// TwinCAT 3 PLC project CleanroomConnect
// ProgramVersion: 3.1.4024.0
// libraries:
//   KMWE Generic Library, * (KMWE)
//   Tc2_MC2, * (Beckhoff Automation GmbH)
//   Tc2_Standard, * (Beckhoff Automation GmbH)
//   Tc2_System, * (Beckhoff Automation GmbH)
//   Tc3_Module, * (Beckhoff Automation GmbH)
//   VisuDialogs, * (System)
//   VisuSymbols,3.5.10.0,System
// project tree:
//   DUTs/ I_Door.TcIO, I_AX5000.TcIO, ST_HmiBottomBar.TcDUT, ST_HmiMiddle.TcDUT, ST_HmiTopBar.TcDUT
//   / E_CtrlState.TcDUT (not stored), E_MODE.TcTLO (not stored), FB_ForceOutput.TcPOU (not stored), F_InRange.TcPOU (not stored), GlobalTextList.TcGTLO, PlcTask.TcTTO, ST_MsgBox.TcDUT (not stored)
//   GVLs/ GVL.TcGVL, GVL_Modules.TcGVL
//   POUs/02 UN/Unit %28UN%29/ ST_UN_CleanroomConnectSettings.TcDUT (not stored), UN_CleanroomConnect.TcPOU (not stored)
//   POUs/03 EM/Equipment %28EM%29/2 EM_PalletConveyor/DUT/ E_SeqCentering.TcDUT (not stored), E_ActionSelection.TcDUT (not stored), E_SeqTransport.TcDUT (not stored)
//   POUs/03 EM/Equipment %28EM%29/2 EM_PalletConveyor/ FB_ModeStateControl_PalletConveyor.TcPOU (not stored) (excluded from build), EM_PalletConveyor.TcPOU (not stored), I_EM_PalletConveyor.TcIO (not stored), ST_SettingsPalletConveyor.TcDUT (not stored)
//   POUs/03 EM/Equipment %28EM%29/4 EM_LiftingTransport/DUT/ E_SeqLiftingTransport.TcDUT (not stored), ST_PositioningProfile.TcDUT (not stored), ST_SettingsLiftingTransport.TcDUT (not stored), ST_SpeedProfile.TcDUT (not stored)
//   POUs/03 EM/Equipment %28EM%29/EM_AirTreatment/DUTs/ I_EM_AirTreatment.TcIO (not stored), ST_SettingsAirTrearment.TcDUT (not stored)
//   POUs/03 EM/Equipment %28EM%29/EM_AirTreatment/ EM_AirTreatment.TcPOU (not stored)
//   POUs/03 EM/Equipment %28EM%29/4 EM_LiftingTransport/ EM_LiftingTransport.TcPOU (not stored), I_EM_LiftingTransport.TcIO (not stored)
//   POUs/03 EM/Equipment %28EM%29/1 EM_Utilities/DUTs/ E_ForceValue.TcDUT (not stored), I_EM_Utilities.TcIO (not stored), ST_SettingsUtilities.TcDUT (not stored)
//   POUs/03 EM/Equipment %28EM%29/1 EM_Utilities/ EM_Utilities.TcPOU (not stored)
//   POUs/03 EM/Equipment %28EM%29/EM_DockingCabin/DUTs/ E_SeqDockingCabin.TcDUT (not stored), ST_SettingsDockingCabin.TcDUT (not stored)
//   POUs/03 EM/Equipment %28EM%29/EM_DockingCabin/ EM_DockingCabin.TcPOU (not stored)
//   POUs/03 EM/Equipment %28EM%29/3 EM_DockingInterface/DUTs/ E_SeqDockingInterface.TcDUT (not stored), I_EM_DockingInterface.TcIO (not stored), ST_SettingsDockingInterface.TcDUT (not stored)
//   POUs/03 EM/Equipment %28EM%29/3 EM_DockingInterface/ EM_DockingInterface.TcPOU (not stored)
//   POUs/03 EM/Equipment %28EM%29/EM_Doors/DUTs/ E_SeqDoors.TcDUT (not stored), I_EM_Doors.TcIO (not stored), ST_SettingsDoors.TcDUT (not stored)
//   POUs/03 EM/Equipment %28EM%29/EM_Doors/ EM_Doors.TcPOU (not stored)
//   POUs/03 EM/ FB_Interlock.TcPOU, FB_InterlockHandler.TcPOU, ST_Interlock.TcDUT (not stored), ST_InterlockList.TcDUT (not stored)
//   POUs/04 CM/Control %28CM%29/CM_AX5000/ CM_AX5000.TcPOU (not stored), E_SeqAX5000.TcDUT (not stored), ST_SettingsAX5000.TcDUT (not stored)
//   POUs/04 CM/Control %28CM%29/CM_DIgitalOutput/ CM_DigOutput.TcPOU (not stored), ST_DigOutput_HMI.TcDUT (not stored)
//   POUs/04 CM/Control %28CM%29/CM_SEW_WithBrake/ CM_SEW_WithBrake.TcPOU (not stored), E_SeqSEW_WithBrake.TcDUT (not stored), ST_SettingsSEW_WithBrake.TcDUT (not stored)
//   POUs/04 CM/Control %28CM%29/CM_MOVITRAC_B/ CM_MOVITRAC_B.TcPOU (not stored), E_SeqMOVITRAC_B_WithBrake.TcDUT (not stored), ST_SettingsMOVITRAC_B_WithBrake.TcDUT (not stored)
//   POUs/04 CM/Control %28CM%29/CM_UnlockingPins/ CM_UnlockingPins.TcPOU (not stored), ST_SettingsUnlockingPins.TcDUT (not stored)
//   POUs/04 CM/Control %28CM%29/CM_DoorLock/ ST_SettingsDoorLock.TcDUT (not stored), CM_DoorLock.TcPOU (not stored)
//   POUs/04 CM/Control %28CM%29/CM_SpeedDoor/ CM_SpeedDoor.TcPOU (not stored), ST_SettingsSpeedDoor.TcDUT (not stored)
//   POUs/04 CM/Control %28CM%29/CM_ValveWithFB/ CM_ValveWithDoubleFB.TcPOU (not stored), CM_ValveWithFB.TcPOU (not stored), ST_SettingsValveWithFB.TcDUT (not stored), ST_ValveWithFB_HMI.TcDUT (not stored)
//   POUs/04 CM/Control %28CM%29/CM_DockingClamps/ CM_DockingClamps.TcPOU (not stored), ST_SettingsDockingClamps.TcDUT (not stored)
//   POUs/04 CM/Control %28CM%29/ E_Location.TcDUT (not stored), FB_Flash.TcPOU (not stored), FB_MovAvg.TcPOU (not stored), FB_Toggle.TcPOU (not stored), I_ServoMotor.TcIO (not stored)
//   POUs/04 CM/Control %28CM%29/OBJ_Carrier/ I_Carrier.TcIO (not stored), OBJ_Carrier.TcPOU (not stored), ST_Carrier.TcDUT (not stored)
//   POUs/ FB_ModeStateControl.TcPOU, FB_ModeStateControl_Base.TcPOU (excluded from build), FB_InRange.TcPOU, MAIN.TcPOU
// real-time tasks:
//   TASK PlcTask: cycle T#10ms, priority 20, ADS port 350
//   TASK PlcTask1: cycle T#10ms, priority 21, ADS port 351
//   TASK VISU_TASK: cycle T#200000us, priority 30, ADS port 352
// motion (NC):
//   TASK NC-Task 1 SAF: cycle T#2ms, priority 4, ADS port 501
//   TASK NC-Task 1 SVB: cycle T#10ms, priority 8, ADS port 511
//   AXIS Lift (id 1)
//     Velo: RefSearch=100, RefSync=10, SlowManual=50, FastManual=100
//     OtherSettings: AllowMotionCmdToSlave=true, PulseDistancePos=10, PulseDistanceNeg=10
//     encoder EncType=1
//       SoftEndMinControl: Enable=true
//       SoftEndMaxControl: Enable=true, Range=500
//       Inc: RefSearchInverse=true, RefSyncInverse=false
//     drive DrvType=5
//       Analog: TorqueSetpointScale=10, ScaleFactorActTorque=0.1
//       TimeComp: TaskDelayCycles=1
//     controller CtrType=1
//       CtrPara: PriorControlFactor=1
//         Observer: BandWidth=20
//   AXIS TransportUnit (id 2)
//     Dynamic: Acceleration=185.271, Deceleration=185.271, Jerk=555.813
//     Velo: RefSearch=1.23514, RefSync=1.23514, SlowManual=0.25, FastManual=1.5, Fast=123.514, Maximum=123.514
//     OtherSettings: AllowMotionCmdToSlave=true
//     encoder EncType=19
//       EncPara: ScaleFactorNumerator=174.487168, ScaleFactorDenominator=52428800, MaxCount=#xffffffff
//         SoftEndMinControl: Enable=true
//         SoftEndMaxControl: Enable=true, Range=1750
//     drive DrvType=16
//       DrvPara: MaxCount=#xffffffff, DriveControlDWord=#x00020100
//         Analog: VeloReferenz=135.8654, VeloScale=32, TorqueSetpointScale=10, ScaleFactorActTorque=0.1
//         TimeComp: TaskDelayCycles=1
//     controller CtrType=1
//       CtrPara: PriorControlFactor=1
//         Observer: BandWidth=20
// I/O:
//   DEVICE Master (EtherCAT) (disabled), AmsNetId 10.130.4.120.2.1
//     Drive 12 (AX5103-0000-0202) [AX5103-0000-0202 EtherCAT Drive (SoE, 1 Ch.)]
//     Term 1 (EK1200) [EK1200-5000 EtherCAT Power supply (2A E-Bus)]
//       Term 2 (EL6070-0033) [EL6070-0033 1Ch. Licence key terminal, individual licences]
//       Term 4 (EL1809) [EL1809 16Ch. Dig. Input 24V, 3ms]
//       Term 5 (EL1809) [EL1809 16Ch. Dig. Input 24V, 3ms]
//       Term 6 (EL1809) [EL1809 16Ch. Dig. Input 24V, 3ms]
//       Term 3 (EL1809) [EL1809 16Ch. Dig. Input 24V, 3ms]
//       Term 7 (EL2809) [EL2809 16Ch. Dig. Output 24V, 0.5A]
//       Term 8 (EL4024) [EL4024 4Ch. Ana. Output 4-20mA, 12bit]
//       Term 17 (EL7211-9014) [EL7211-9014 1Ch. MDP742 Servo motor output stage with OCT (50V, 4.5A RMS) and STO input]
//         startup 32786:19 := 0000 // DRV Brake Settings / Emergency application timeout
//         startup 32784:51 := 0A00 // DRV Amplifier Settings / Stand still window
//         startup 32785:27 := 4F080000 // DRV Motor Settings / Motor speed limitation
//         startup 28688:11 := D007 // Torque limitation
//         startup 32784:19 := 8701 // DRV Amplifier Settings / Current loop proportional gain
//         startup 32784:18 := 0500 // DRV Amplifier Settings / Current loop integral time
//         startup 32784:21 := 6A030000 // DRV Amplifier Settings / Velocity loop proportional gain
//         startup 32784:20 := 96000000 // DRV Amplifier Settings / Velocity loop integral time
//         startup 32768:1 := 00 // FB Settings / Invert feedback direction
//       Term 9 (EL9110) [EL9110 Power Supplier with LED (24V, Diagnostics)]
//       Term 10 (EL2809) [EL2809 16Ch. Dig. Output 24V, 0.5A]
//       Term 11 (EL9011) [EL9011 End Terminal]
//   DEVICE Device 2 (EtherCAT) (disabled), AmsNetId 10.130.4.120.3.1
//     Term 15 (EK1200) [EK1200-5000 EtherCAT Power supply (2A E-Bus)]
//       Term 16 (EL6070-0033) [EL6070-0033 1Ch. Licence key terminal, individual licences]
//       Term 18 (EL1904) [EL1904, 4 Ch. Safety Input 24V, TwinSAFE]
//         modules: Module 1 (FSOES)
//       Term 19 (EL1904) [EL1904, 4 Ch. Safety Input 24V, TwinSAFE]
//         modules: Module 1 (FSOES)
//       Term 23 (EL1918) [EL1918, 8Ch. Safety Input 24V, TwinSAFE]
//         modules: Module 1 (FSOE), Module 2 (FSLOGIC)
//       Term 22 (EL2904) [EL2904, 4 Ch. Safety Output 24V, 0.5A, TwinSAFE]
//         modules: Module 1 (FSOES), Module 2 (DO)
//       Term 24 (AX5805) [AX5805 (Safety Drive Option)]
//         modules: Module 1 (Safety Process Data, 2 axis), Module 2 (Standard Process Data, 2 axis)
// variable links:
//   NC-Task 1 SAF/Axes/TransportUnit <-> Master (EtherCAT)/Term 1 (EK1200)/Term 17 (EL7211-9014)
//     Drive/Inputs/In/nDataIn1 <-> DRV Following error actual value/Following error actual value
//     Drive/Inputs/In/nDcOutputTime <-> InfoData/DcOutputShift
//     Drive/Inputs/In/nState1 <-> DRV Statusword/Statusword
//     Drive/Inputs/In/nState2 <-> DRV Statusword/Statusword @bit 8
//     Drive/Inputs/In/nState4 @bit 1 <-> WcState/InputToggle
//     Drive/Inputs/In/nState4 <-> WcState/WcState
//     Drive/Outputs/Out/nCtrl1 <-> DRV Controlword/Controlword
//     Drive/Outputs/Out/nCtrl2 <-> DRV Controlword/Controlword @bit 8
//     Drive/Outputs/Out/nDataOut1 <-> DRV Target position/Target position
//     Drive/Outputs/Out/nDataOut2 <-> DRV Target velocity/Target velocity
//     Drive/Outputs/Out/nDataOut4 <-> DRV Target torque/Target torque
//     Enc/Inputs/In/nDataIn1 <-> FB Position/Position
//     Enc/Inputs/In/nDataIn4 <-> FB Touch probe 1 neg position/TP1 Neg position
//     Enc/Inputs/In/nDataIn6 <-> FB Touch probe 2 neg position/TP2 Neg position
//     Enc/Inputs/In/nDcInputTime <-> InfoData/DcInputShift
//     Enc/Inputs/In/nState4 @bit 1 <-> WcState/InputToggle
//     Enc/Inputs/In/nState4 <-> WcState/WcState
//     Enc/Inputs/In/nState5 <-> FB Touch probe status/Touch probe status/TP1 Enable
//     Enc/Inputs/In/nState6 <-> FB Touch probe status/Touch probe status/TP2 Enable
//     Enc/Inputs/In/nState5 @bit 7 <-> FB Touch probe status/Touch probe status/TP1 Input
//     Enc/Inputs/In/nState6 @bit 7 <-> FB Touch probe status/Touch probe status/TP2 Input
//     Enc/Inputs/In/nState5 @bit 2 <-> FB Touch probe status/Touch probe status/TP1 Neg value stored
//     Enc/Inputs/In/nState6 @bit 2 <-> FB Touch probe status/Touch probe status/TP2 Neg value stored
//     Enc/Inputs/In/nState5 @bit 1 <-> FB Touch probe status/Touch probe status/TP1 Pos value stored
//     Enc/Inputs/In/nState6 @bit 1 <-> FB Touch probe status/Touch probe status/TP2 Pos value stored
//     Enc/Outputs/Out/nCtrl5 @bit 1 <-> FB Touch probe control/Touch probe function/TP1 Continous
//     Enc/Outputs/Out/nCtrl6 @bit 1 <-> FB Touch probe control/Touch probe function/TP2 Continous
//     Enc/Outputs/Out/nCtrl5 <-> FB Touch probe control/Touch probe function/TP1 Enable
//     Enc/Outputs/Out/nCtrl6 <-> FB Touch probe control/Touch probe function/TP2 Enable
//     Enc/Outputs/Out/nCtrl5 @bit 5 <-> FB Touch probe control/Touch probe function/TP1 Enable neg edge
//     Enc/Outputs/Out/nCtrl6 @bit 5 <-> FB Touch probe control/Touch probe function/TP2 Enable neg edge
//     Enc/Outputs/Out/nCtrl5 @bit 4 <-> FB Touch probe control/Touch probe function/TP1 Enable pos edge
//     Enc/Outputs/Out/nCtrl6 @bit 4 <-> FB Touch probe control/Touch probe function/TP2 Enable pos edge
//     Enc/Outputs/Out/nCtrl5 @bit 2 <-> FB Touch probe control/Touch probe function/TP1 Trigger mode
//     Enc/Outputs/Out/nCtrl6 @bit 2 <-> FB Touch probe control/Touch probe function/TP2 Trigger mode
//   CleanroomConnect/CleanroomConnect Instance <-> HardwareSimulator/HardwareSimulator Instance
//     PlcTask Inputs/GVL_Modules.g_emDockingInterface.s_cmDockingClampsLower.I_bStaValveIsOff <-> PlcTask Outputs/MAIN.simDockingClampLower.Q_bStaFeedbackOff
//     PlcTask Inputs/GVL_Modules.g_emDockingInterface.s_cmDockingClampsLower.I_bStaValveIsOff2 <-> PlcTask Outputs/MAIN.simDockingClampLower.Q_bStaFeedbackOff2
//     PlcTask Inputs/GVL_Modules.g_emDockingInterface.s_cmDockingClampsLower.I_bStaValveIsOn <-> PlcTask Outputs/MAIN.simDockingClampLower.Q_bStaFeedbackOn
//     PlcTask Inputs/GVL_Modules.g_emDockingInterface.s_cmDockingClampsLower.I_bStaValveIsOn2 <-> PlcTask Outputs/MAIN.simDockingClampLower.Q_bStaFeedbackOn2
//     PlcTask Inputs/GVL_Modules.g_emDockingInterface.s_cmDockingClampsUpper.I_bStaValveIsOff <-> PlcTask Outputs/MAIN.simDockingClampUpper.Q_bStaFeedbackOff
//     PlcTask Inputs/GVL_Modules.g_emDockingInterface.s_cmDockingClampsUpper.I_bStaValveIsOff2 <-> PlcTask Outputs/MAIN.simDockingClampUpper.Q_bStaFeedbackOff2
//     PlcTask Inputs/GVL_Modules.g_emDockingInterface.s_cmDockingClampsUpper.I_bStaValveIsOn <-> PlcTask Outputs/MAIN.simDockingClampUpper.Q_bStaFeedbackOn
//     PlcTask Inputs/GVL_Modules.g_emDockingInterface.s_cmDockingClampsUpper.I_bStaValveIsOn2 <-> PlcTask Outputs/MAIN.simDockingClampUpper.Q_bStaFeedbackOn2
//     PlcTask Inputs/GVL_Modules.g_emDockingInterface.s_cmDoorOpener.I_bStaValveIsOff <-> PlcTask Outputs/MAIN.simDoorOpener.Q_bStaFeedbackOff
//     PlcTask Inputs/GVL_Modules.g_emDockingInterface.s_cmDoorOpener.I_bStaValveIsOn <-> PlcTask Outputs/MAIN.simDoorOpener.Q_bStaFeedbackOn
//     PlcTask Inputs/GVL_Modules.g_emDockingInterface.s_cmDoorShutter.I_bStaValveIsOff <-> PlcTask Outputs/MAIN.simDoorShutter.Q_bStaFeedbackOff
//     PlcTask Inputs/GVL_Modules.g_emDockingInterface.s_cmDoorShutter.I_bStaValveIsOn <-> PlcTask Outputs/MAIN.simDoorShutter.Q_bStaFeedbackOn
//     PlcTask Inputs/GVL_Modules.g_emDockingInterface.s_cmUnlockingPinLower.I_bStaValveIsOff <-> PlcTask Outputs/MAIN.simUnlockPinLower.Q_bStaFeedbackOff
//     PlcTask Inputs/GVL_Modules.g_emDockingInterface.s_cmUnlockingPinLower.I_bStaValveIsOn <-> PlcTask Outputs/MAIN.simUnlockPinLower.Q_bStaFeedbackOn
//     PlcTask Inputs/GVL_Modules.g_emDockingInterface.s_cmUnlockingPinUpper.I_bStaValveIsOff <-> PlcTask Outputs/MAIN.simUnlockPinUpper.Q_bStaFeedbackOff
//     PlcTask Inputs/GVL_Modules.g_emDockingInterface.s_cmUnlockingPinUpper.I_bStaValveIsOn <-> PlcTask Outputs/MAIN.simUnlockPinUpper.Q_bStaFeedbackOn
//     PlcTask Inputs/GVL_Modules.g_emDockingInterface.s_diStaDoorAlmostClosed.I_bStaInput <-> PlcTask Outputs/MAIN.simDoorOpenerAlmostClosed
//     PlcTask Inputs/GVL_Modules.g_emPalletConveyor.s_cmCenteringUnit.I_bStaValveIsOff <-> PlcTask Outputs/MAIN.simCentering.Q_bStaFeedbackOff
//     PlcTask Inputs/GVL_Modules.g_emPalletConveyor.s_cmCenteringUnit.I_bStaValveIsOff2 <-> PlcTask Outputs/MAIN.simCentering.Q_bStaFeedbackOff2
//     PlcTask Inputs/GVL_Modules.g_emPalletConveyor.s_cmCenteringUnit.I_bStaValveIsOn <-> PlcTask Outputs/MAIN.simCentering.Q_bStaFeedbackOn
//     PlcTask Inputs/GVL_Modules.g_emPalletConveyor.s_cmCenteringUnit.I_bStaValveIsOn2 <-> PlcTask Outputs/MAIN.simCentering.Q_bStaFeedbackOn2
//     PlcTask Inputs/GVL_Modules.g_emPalletConveyor.s_cmPalletConveyor.I_bStaMotorIsRunning <-> PlcTask Outputs/MAIN.sim_MOVITRAC_B.Q_bStaMotorIsRunning
//     PlcTask Inputs/GVL_Modules.g_emPalletConveyor.s_cmPalletConveyor.I_bStaReadyForOperation <-> PlcTask Outputs/MAIN.sim_MOVITRAC_B.Q_bStaReadyForOperation
//     PlcTask Inputs/GVL_Modules.g_emUtilities.s_diAirPressureOk.I_bStaInput <-> PlcTask Outputs/MAIN.simAirPressureOK
//     PlcTask Inputs/GVL_Modules.g_emUtilities.s_diPower400VacOk.I_bStaInput <-> PlcTask Outputs/MAIN.simPowerOK
//     PlcTask Inputs/GVL_Modules.g_emUtilities.s_diSafetyOk.I_bStaInput <-> PlcTask Outputs/MAIN.simSafetyOK
//     PlcTask Outputs/GVL_Modules.g_emDockingInterface.s_cmDockingClampsLower.Q_bCmdOff <-> PlcTask Inputs/MAIN.simDockingClampLower.I_bCmdValveOff
//     PlcTask Outputs/GVL_Modules.g_emDockingInterface.s_cmDockingClampsLower.Q_bCmdOn <-> PlcTask Inputs/MAIN.simDockingClampLower.I_bCmdValveOn
//     PlcTask Outputs/GVL_Modules.g_emDockingInterface.s_cmDockingClampsUpper.Q_bCmdOff <-> PlcTask Inputs/MAIN.simDockingClampUpper.I_bCmdValveOff
//     PlcTask Outputs/GVL_Modules.g_emDockingInterface.s_cmDockingClampsUpper.Q_bCmdOn <-> PlcTask Inputs/MAIN.simDockingClampUpper.I_bCmdValveOn
//     PlcTask Outputs/GVL_Modules.g_emDockingInterface.s_cmDoorOpener.Q_bCmdOff <-> PlcTask Inputs/MAIN.simDoorOpener.I_bCmdValveOff
//     PlcTask Outputs/GVL_Modules.g_emDockingInterface.s_cmDoorOpener.Q_bCmdOn <-> PlcTask Inputs/MAIN.simDoorOpener.I_bCmdValveOn
//     PlcTask Outputs/GVL_Modules.g_emDockingInterface.s_cmDoorShutter.Q_bCmdOff <-> PlcTask Inputs/MAIN.simDoorShutter.I_bCmdValveOff
//     PlcTask Outputs/GVL_Modules.g_emDockingInterface.s_cmDoorShutter.Q_bCmdOn <-> PlcTask Inputs/MAIN.simDoorShutter.I_bCmdValveOn
//     PlcTask Outputs/GVL_Modules.g_emDockingInterface.s_cmUnlockingPinLower.Q_bCmdOff <-> PlcTask Inputs/MAIN.simUnlockPinLower.I_bCmdValveOff
//     PlcTask Outputs/GVL_Modules.g_emDockingInterface.s_cmUnlockingPinLower.Q_bCmdOn <-> PlcTask Inputs/MAIN.simUnlockPinLower.I_bCmdValveOn
//     PlcTask Outputs/GVL_Modules.g_emDockingInterface.s_cmUnlockingPinUpper.Q_bCmdOff <-> PlcTask Inputs/MAIN.simUnlockPinUpper.I_bCmdValveOff
//     PlcTask Outputs/GVL_Modules.g_emDockingInterface.s_cmUnlockingPinUpper.Q_bCmdOn <-> PlcTask Inputs/MAIN.simUnlockPinUpper.I_bCmdValveOn
//     PlcTask Outputs/GVL_Modules.g_emPalletConveyor.s_cmCenteringUnit.Q_bCmdOff <-> PlcTask Inputs/MAIN.simCentering.I_bCmdValveOff
//     PlcTask Outputs/GVL_Modules.g_emPalletConveyor.s_cmCenteringUnit.Q_bCmdOn <-> PlcTask Inputs/MAIN.simCentering.I_bCmdValveOn
//     PlcTask Outputs/GVL_Modules.g_emPalletConveyor.s_cmPalletConveyor.Q_bCmdEnable <-> PlcTask Inputs/MAIN.sim_MOVITRAC_B.I_bCmdEnable
//     PlcTask Outputs/GVL_Modules.g_emPalletConveyor.s_cmPalletConveyor.Q_bCmdReset <-> PlcTask Inputs/MAIN.sim_MOVITRAC_B.I_bCmdReset
//     PlcTask Outputs/GVL_Modules.g_emPalletConveyor.s_cmPalletConveyor.Q_bCmdStartCCW <-> PlcTask Inputs/MAIN.sim_MOVITRAC_B.I_bCmdStartCCW
//     PlcTask Outputs/GVL_Modules.g_emPalletConveyor.s_cmPalletConveyor.Q_bCmdStartCW <-> PlcTask Inputs/MAIN.sim_MOVITRAC_B.I_bCmdStartCW

CONFIGURATION CleanroomConnect
    RESOURCE PLC ON TwinCAT3
        TASK PlcTask(INTERVAL := T#10ms, PRIORITY := 20);
        PROGRAM MAIN WITH PlcTask : MAIN;
    END_RESOURCE
END_CONFIGURATION

// ---- DUTs/ST_HmiBottomBar.TcDUT
TYPE ST_HmiBottomBar :
STRUCT CONSTANT 
	Start					: STRING := 'Bottom/BottomBar_Start.Content';
	General_ReturnToStart	: STRING := 'Bottom/BottomBar_ReturnToStart.Content';
	General_Return			: STRING := 'Bottom/BottomBar_Return.Content';
	Alarm					: STRING := 'Bottom/BottomBar_AlarmManager.Content';
	Procedure				: STRING := 'Bottom/BottomBar_Procedure.Content';
END_STRUCT
END_TYPE

// ---- DUTs/ST_HmiMiddle.TcDUT
TYPE ST_HmiMiddle :
STRUCT CONSTANT 
	
	//--------------------------------//
	//General Pages
	Start								: STRING 	:= 'WebContent/Middle/Start.content';
	AlarmManager						: STRING	:= 'WebContent/Middle/AlarmManager.content';
	ParameterManager					: STRING	:= 'WebContent/Middle/ParameterManager.content';

	//Equipment Modules
	EM_Utilities						: STRING	:= 'WebContent/Middle/EM_Utilities/EM_Utilities.content';
	EM_PalletConveyor					: STRING	:= 'WebContent/Middle/EM_PalletConveyor/EM_PalletConveyor.content';	
	EM_DockingInterface					: STRING	:= 'WebContent/Middle/EM_DockingInterface/EM_DockingInterface.content';
	EM_LiftingTransport					: STRING	:= 'WebContent/Middle/EM_LiftingTransport/EM_LiftingTransport.content';
	EM_Cabin							: STRING	:= 'WebContent/Middle/EM_Cabin/EM_Cabin.content';
	EM_Doors							: STRING	:= 'WebContent/Middle/EM_Doors/EM_Doors.content';
	//..
	//..
	
	
	//--TesterConfig						: STRING	:= 'Middle/TesterConfig.Content';
	//--PPLSelection						: STRING	:= 'Middle/PPLSelection.Content';
	//--AlarmManager						: STRING	:= 'Middle/AlarmManager.Content';
	//--Procedures							: STRING	:= 'Middle/Procedures.Content';
	//--ProcedureStart						: STRING	:= 'Middle/ProceduresStart.Content';
	//--ProceduresCalibration				: STRING	:= 'Middle/ProceduresCalibration.Content';
	//--Manual								: STRING	:= 'Middle/Manual.Content';
	//--------------------------------//
	
	//--------------------------------//
	//MagneticTest
	//--OperatorInputData					: STRING	:= 'Middle/MagneticTest/OperatorInputData.Content';
	//--OperatorPrepareTester				: STRING	:= 'Middle/MagneticTest/OperatorPrepareTester.Content';
	//--ProcedureTesting					: STRING	:= 'Middle/MagneticTest/ProcedureTesting.Content';
	//--OperatorDisconnect					: STRING	:= 'Middle/MagneticTest/OperatorDisconnect.Content';
	//--OperatorMoveDown					: STRING	:= 'Middle/MagneticTest/OperatorMoveDown.Content';
	//--------------------------------//
	

END_STRUCT
END_TYPE

// ---- DUTs/ST_HmiTopBar.TcDUT
TYPE ST_HmiTopBar :
STRUCT CONSTANT 
	GeneralTopbar	: STRING := 'Top/TopBar.Content';
END_STRUCT
END_TYPE

// ---- GVLs/GVL.TcGVL
{attribute 'qualified_only'}
VAR_GLOBAL
	g_unCleanroomConnect		: UN_CleanroomConnect;
	
	g_eStaLedColor 				: E_KmweLedColors := E_KmweLedColors.Idle;
	g_bLedFlashSlow 			: BOOL;
	g_bLedFlashFast				: BOOL;

	g_fbHmiBtnSimulation		: FB_HmiBtn;
	
	g_sUser						: STRING;
	g_sSerialNumber				: STRING;
	g_sNotesEntry				: T_MAXSTRING;
	
	//Hmi linked variable
	g_sToHmiTopContent			: STRING;
	g_sToHmiMiddleContent		: STRING;
	g_sToHmiBottomContent		: STRING;
	
	//Structs with screens that can be appointed to linked variables
	g_stHmiTopBar				: ST_HmiTopBar;
	g_stHmiMiddle				: ST_HmiMiddle;
	g_stHmiBottomBar			: ST_HmiBottomBar;
	
	g_osrNotify					: R_TRIG;	
END_VAR

VAR_GLOBAL CONSTANT
	g_MAX_LEN_INTERLOCK_REASON : USINT := 64;
	g_LEN_INTERLOCK_LIST : USINT := 5;
END_VAR

// ---- GVLs/GVL_Modules.TcGVL
{attribute 'qualified_only'}
VAR_GLOBAL
	g_emUtilities : EM_Utilities;
	g_emPalletConveyor : EM_PalletConveyor;
	g_emDockingInterface : EM_DockingInterface;
//##_LIFTING_TRANSPORT_DISABLED_##	g_emLiftingTransport : EM_LiftingTransport;
//##_DOCKING_CABIN_DISABLED_##	g_emDockingCabin : EM_DockingCabin;
//##_DOORS_DISABLED_##	g_emDoors : EM_Doors;
	
	g_objCarrier : OBJ_Carrier;
END_VAR

// ---- DUTs/I_Door.TcIO
INTERFACE I_Door
VAR_INPUT
	bEnable : BOOL;
	bEnablePositive : BOOL; 
	bEnableNegative : BOOL;
END_VAR

METHOD PUBLIC m_Close : BOOL
END_METHOD

METHOD PUBLIC m_Open : BOOL
END_METHOD

METHOD PUBLIC m_Reset : BOOL
END_METHOD

METHOD PUBLIC m_Stop : BOOL
END_METHOD

{attribute 'monitoring':='call'}
PROPERTY PUBLIC p_bStaIsClosed : BOOL
GET
END_GET
END_PROPERTY

{attribute 'monitoring':='call'}
PROPERTY PUBLIC p_bStaIsClosing : BOOL
GET
END_GET
END_PROPERTY

{attribute 'monitoring':='call'}
PROPERTY PUBLIC p_bStaIsOpened : BOOL
GET
END_GET
END_PROPERTY

{attribute 'monitoring':='call'}
PROPERTY PUBLIC p_bStaIsOpening : BOOL
GET
END_GET
END_PROPERTY

END_INTERFACE

// ---- DUTs/I_AX5000.TcIO
INTERFACE I_AX5000

METHOD PUBLIC m_MC_Home : BOOL
VAR_INPUT
	i_bExecute : BOOL;
	i_fPosition : REAL;
	i_eHomingMode : TC2_MC2.MC_HomingMode;
	i_eBufferMode : TC2_MC2.MC_BufferMode;
END_VAR
END_METHOD

METHOD PUBLIC m_MC_Jog : BOOL
VAR_INPUT
	i_bExecute : BOOL;
	i_bJogForward : BOOL;
	i_bJogBackward : BOOL;
	i_eJogMode : TC2_MC2.E_JogMode;
	i_fPosition : LREAL; 
	i_fVelocity : LREAL; 
	i_fAcceleration : LREAL; 
	i_fDeceleration : LREAL; 
	i_fJerk : LREAL;
END_VAR
END_METHOD

METHOD PUBLIC m_MC_MoveAbsolute : BOOL
VAR_INPUT
	i_bExecute : BOOL;
	i_fPosition : LREAL; 
	i_fVelocity : LREAL; 
	i_fAcceleration : LREAL; 
	i_fDeceleration : LREAL; 
	i_fJerk : LREAL;
	i_eBufferMode : TC2_MC2.MC_BufferMode;
END_VAR
END_METHOD

METHOD PUBLIC m_MC_MoveRelative : BOOL
VAR_INPUT
	i_bExecute : BOOL;
	i_fDistance : LREAL; 
	i_fVelocity : LREAL; 
	i_fAcceleration : LREAL; 
	i_fDeceleration : LREAL; 
	i_fJerk : LREAL;
	i_eBufferMode : TC2_MC2.MC_BufferMode;
END_VAR
END_METHOD

METHOD PUBLIC m_MC_MoveVelocity : BOOL
VAR_INPUT
	i_bExecute : BOOL;
	i_fVelocity : LREAL; 
	i_fAcceleration : LREAL; 
	i_fDeceleration : LREAL; 
	i_fJerk : LREAL;
	i_eDirection : TC2_MC2.MC_Direction;
	i_eBufferMode : TC2_MC2.MC_BufferMode;
END_VAR
END_METHOD

METHOD PUBLIC m_MC_Power : BOOL
VAR_INPUT
	i_bEnable : BOOL;
	i_bEnablePositive : BOOL;
	i_bEnableNegative : BOOL;
	i_fOverride : LREAL;
	i_eBufferMode : TC2_MC2.MC_BufferMode;
END_VAR
END_METHOD

METHOD PUBLIC m_MC_Reset : BOOL
VAR_INPUT
	i_bExecute : BOOL;
END_VAR
END_METHOD

METHOD PUBLIC m_MC_Stop : BOOL
VAR_INPUT
	i_bExecute : BOOL;
	i_fDeceleration : LREAL;
	i_fJerk : LREAL;
END_VAR
END_METHOD

PROPERTY PUBLIC p_bActive : BOOL
GET
END_GET
END_PROPERTY

PROPERTY PUBLIC p_bBusy : BOOL
GET
END_GET
END_PROPERTY

PROPERTY PUBLIC p_bCommandAborted : BOOL
GET
END_GET
END_PROPERTY

PROPERTY PUBLIC p_bDone : BOOL
GET
END_GET
END_PROPERTY

PROPERTY PUBLIC p_bError : BOOL
GET
END_GET
END_PROPERTY

PROPERTY PUBLIC p_bHomed : BOOL
GET
END_GET
END_PROPERTY

PROPERTY PUBLIC p_bInVelocity : BOOL
GET
END_GET
END_PROPERTY

PROPERTY PUBLIC p_bStandstill : BOOL
GET
END_GET
END_PROPERTY

PROPERTY PUBLIC p_fPosition : LREAL
GET
END_GET
END_PROPERTY

PROPERTY PUBLIC p_fVelocity : LREAL
GET
END_GET
END_PROPERTY

PROPERTY PUBLIC p_nErrorID : UDINT
GET
END_GET
END_PROPERTY

END_INTERFACE

// ---- POUs/MAIN.TcPOU
PROGRAM MAIN
VAR
	s_ParamPathnames	: ARRAY[1..Param_Project.n_MaxParamFolders] OF STRING := ['C:\Cleanroom_Connect\Parameters'];//, 'C:\Cleanroom_Connect\Param\DockingInterface'];

	User : STRING := '<user_name>';
	SoftwareVersion : STRING := '<software_version>';
	InitDone : BOOL;
	Shutdown : BOOL;
	
	fTestValue : LREAL; 
	
	stMsgBox : ST_MsgBox;
	
	fbModeStateControl : FB_ModeStateControl;
	
	//Test other valv configuration (2x 3/2 vs 1x 5/3 with open middle position)	
	Q_bTestDoorShutterClose AT%Q* : BOOL;	//Link to: Output . Channel 15 . K21 (EL2809) . Master (EtherCAT) . Devices
	Q_bTestDoorShutterOpen AT%Q* : BOOL;	//Link to: Output . Channel 16 . K21 (EL2809) . Master (EtherCAT) . Devices
	s_tofPressurizeDelay : TOF;
	s_nCmd : UINT; // 0 = IDLE, 1 = CLOSE, 2 = OPEN 
	
	
END_VAR

GVL_KMWEGenericLib.g_fbAlarmManager();


GVL_KMWEGenericLib.g_fbParamManager.p_bShowHmiParam := TRUE;

GVL_KMWEGenericLib.g_fbParamManager(
	i_sPathName := s_ParamPathnames, 
	i_osrResetImportExport := GVL_KMWEGenericLib.g_fbAlarmManager.p_osrReset);

fbModeStateControl();
	
GVL.g_unCleanroomConnect.p_bCmdReset := GVL_KMWEGenericLib.g_fbAlarmManager.p_osrReset;
GVL.g_unCleanroomConnect();


{warning '#TEST: Code below is just test code for a quick test, can be removed if no longer after  test is finisched'}
(*
s_tofPressurizeDelay(IN := s_nCmd = 0, PT := T#75mS);

CASE s_nCmd OF
	0: //IDLE
		Q_bTestDoorShutterClose := TRUE;
		Q_bTestDoorShutterOpen := TRUE;
		
	1: //CLOSE
		Q_bTestDoorShutterOpen := NOT s_tofPressurizeDelay.Q;
		Q_bTestDoorShutterClose := FALSE;
	
	2: //OPEN
		Q_bTestDoorShutterClose := NOT s_tofPressurizeDelay.Q;
		Q_bTestDoorShutterOpen := FALSE;

END_CASE
*)

END_PROGRAM

// ---- POUs/FB_ModeStateControl.TcPOU
FUNCTION_BLOCK FB_ModeStateControl //EXTENDS FB_ModeStateControl_Base
VAR_INPUT
	i_bReqStopAlarm	: BOOL;
	i_bStaAllStopped : BOOL;
END_VAR
VAR_OUTPUT
END_VAR
VAR
	s_bInitDone : BOOL := FALSE;	

	s_eCtrlMode : E_CtrlMode := E_CtrlMode.IDLE;
	s_eCtrlState : E_CtrlState := E_CtrlState.STOPPED;
	
	s_fbHmiBtnModeAutomatic : FB_HmiBtn;
	s_fbHmiBtnModeManual : FB_HmiBtn;
	s_fbHmiBtnModeMaintenance : FB_HmiBtn;
	s_fbHmiBtnModeIO : FB_HmiBtn;
	s_fbHmiBtnModeCleaning : FB_HmiBtn;
	
	s_fbHmiBtnStateStart : FB_HmiBtn;
	s_fbHmiBtnStateStop : FB_HmiBtn;
	s_fbHmiBtnStateReset : FB_HmiBtn;
END_VAR


m_Main();

METHOD PROTECTED _m_Devices : BOOL

//Mode buttons
s_fbHmiBtnModeAutomatic();
s_fbHmiBtnModeManual();
s_fbHmiBtnModeMaintenance();
s_fbHmiBtnModeIO();
s_fbHmiBtnModeCleaning();

//State buttons
s_fbHmiBtnStateStart();
s_fbHmiBtnStateStop();
s_fbHmiBtnStateReset();

CASE s_eCtrlMode OF
	E_CtrlMode.IDLE:
		s_fbHmiBtnModeAutomatic.p_bStaVisible := TRUE;
		s_fbHmiBtnModeManual.p_bStaVisible := TRUE;
		s_fbHmiBtnModeMaintenance.p_bStaVisible := TRUE;
		s_fbHmiBtnModeIO.p_bStaVisible := TRUE;
		s_fbHmiBtnModeCleaning.p_bStaVisible := TRUE;
	
		s_fbHmiBtnStateStart.p_bStaVisible := TRUE;
		s_fbHmiBtnStateStop.p_bStaVisible := TRUE;
		s_fbHmiBtnStateReset.p_bStaVisible := TRUE;
	
	E_CtrlMode.AUTOMATIC:
		;
	
	E_CtrlMode.MANUAL:
		;
	
	E_CtrlMode.MAINTENANCE:
		;
	
	E_CtrlMode.IO:
		;
		
	E_CtrlMode.CLEANING:
		;
	ELSE
		s_eCtrlMode := E_CtrlMode.IDLE;
END_CASE

IF (s_eCtrlState = E_CtrlState.STOPPED) OR (s_eCtrlState = E_CtrlState.IDLE) THEN
		IF s_fbHmiBtnModeAutomatic.p_osrBtnPress THEN
			s_eCtrlMode := E_CtrlMode.AUTOMATIC;

		ELSIF s_fbHmiBtnModeManual.p_osrBtnPress THEN			
			s_eCtrlMode := E_CtrlMode.MANUAL;
		
		ELSIF s_fbHmiBtnModeMaintenance.p_osrBtnPress THEN
			s_eCtrlMode := E_CtrlMode.MAINTENANCE;
		
		ELSIF s_fbHmiBtnModeIO.p_osrBtnPress THEN
			s_eCtrlMode := E_CtrlMode.IO;
		
		ELSIF s_fbHmiBtnModeCleaning.p_osrBtnPress THEN
			s_eCtrlMode := E_CtrlMode.CLEANING;
			
		END_IF
	END_IF

CASE s_eCtrlState OF
	
	E_CtrlState.STOPPED:
	
		IF s_fbHmiBtnStateReset.p_osrBtnPress THEN
			s_eCtrlState := E_CtrlState.IDLE;
		END_IF 
	
	E_CtrlState.IDLE:
	
		IF s_fbHmiBtnStateStop.p_osrBtnPress THEN
			s_eCtrlState := E_CtrlState.STOPPING;
		ELSIF s_fbHmiBtnStateStart.p_osrBtnPress THEN
			s_eCtrlState := E_CtrlState.RUNNING;
		END_IF
			
	E_CtrlState.RUNNING:
	
		IF s_fbHmiBtnStateStop.p_osrBtnPress OR i_bReqStopAlarm THEN
			s_eCtrlState := E_CtrlState.STOPPING;
		END_IF
	
	E_CtrlState.STOPPING:
	
		IF i_bStaAllStopped THEN
			s_eCtrlState := E_CtrlState.STOPPED;
		END_IF
		
ELSE
	s_eCtrlState := E_CtrlState.STOPPED;
END_CASE

IF (s_eCtrlState = E_CtrlState.IDLE) OR (s_eCtrlState = E_CtrlState.STOPPED) THEN
	s_fbHmiBtnModeAutomatic.p_bStaEnabled := s_eCtrlMode <> E_CtrlMode.AUTOMATIC;
	s_fbHmiBtnModeManual.p_bStaEnabled := s_eCtrlMode <> E_CtrlMode.MANUAL;
	s_fbHmiBtnModeMaintenance.p_bStaEnabled := s_eCtrlMode <> E_CtrlMode.MAINTENANCE;
	s_fbHmiBtnModeIO.p_bStaEnabled := s_eCtrlMode <> E_CtrlMode.IO;
	s_fbHmiBtnModeCleaning.p_bStaEnabled := s_eCtrlMode <> E_CtrlMode.CLEANING;
ELSE
	s_fbHmiBtnModeAutomatic.p_bStaEnabled := FALSE;
	s_fbHmiBtnModeManual.p_bStaEnabled := FALSE;
	s_fbHmiBtnModeMaintenance.p_bStaEnabled := FALSE;
	s_fbHmiBtnModeIO.p_bStaEnabled := FALSE;
	s_fbHmiBtnModeCleaning.p_bStaEnabled := FALSE;
END_IF

IF (s_eCtrlMode <> E_CtrlMode.IDLE) THEN
	s_fbHmiBtnStateStart.p_bStaEnabled := s_eCtrlState = E_CtrlState.IDLE;
	s_fbHmiBtnStateStop.p_bStaEnabled := s_eCtrlState = E_CtrlState.RUNNING OR s_eCtrlState = E_CtrlState.IDLE;
	s_fbHmiBtnStateReset.p_bStaEnabled := s_eCtrlState = E_CtrlState.STOPPED;
ELSE
	s_fbHmiBtnStateStart.p_bStaEnabled := FALSE;
	s_fbHmiBtnStateStop.p_bStaEnabled := FALSE;
	s_fbHmiBtnStateReset.p_bStaEnabled := FALSE;
END_IF

_m_Devices := TRUE;
END_METHOD

METHOD PROTECTED _m_Init : BOOL

//Mode buttons
s_fbHmiBtnModeAutomatic.p_eButtontype := E_HmiButtonType.PUSHBUTTON;
s_fbHmiBtnModeAutomatic.p_bStaVisible := FALSE;
s_fbHmiBtnModeAutomatic.p_bStaEnabled := FALSE;
s_fbHmiBtnModeAutomatic.p_sBtnText := 'Automatic';

s_fbHmiBtnModeManual.p_eButtontype := E_HmiButtonType.PUSHBUTTON;
s_fbHmiBtnModeManual.p_bStaVisible := FALSE;
s_fbHmiBtnModeManual.p_bStaEnabled := FALSE;
s_fbHmiBtnModeManual.p_sBtnText := 'Manual';

s_fbHmiBtnModeMaintenance.p_eButtontype := E_HmiButtonType.PUSHBUTTON;
s_fbHmiBtnModeMaintenance.p_bStaVisible := FALSE;
s_fbHmiBtnModeMaintenance.p_bStaEnabled := FALSE;
s_fbHmiBtnModeMaintenance.p_sBtnText := 'Maintenance';

s_fbHmiBtnModeIO.p_eButtontype := E_HmiButtonType.PUSHBUTTON;
s_fbHmiBtnModeIO.p_bStaVisible := FALSE;
s_fbHmiBtnModeIO.p_bStaEnabled := FALSE;
s_fbHmiBtnModeIO.p_sBtnText := 'IO';

s_fbHmiBtnModeCleaning.p_eButtontype := E_HmiButtonType.PUSHBUTTON;
s_fbHmiBtnModeCleaning.p_bStaVisible := FALSE;
s_fbHmiBtnModeCleaning.p_bStaEnabled := FALSE;
s_fbHmiBtnModeCleaning.p_sBtnText := 'Cleaning';

//State buttons
s_fbHmiBtnStateStart.p_eButtontype := E_HmiButtonType.PUSHBUTTON;
s_fbHmiBtnStateStart.p_bStaVisible := FALSE;
s_fbHmiBtnStateStart.p_bStaEnabled := FALSE;
s_fbHmiBtnStateStart.p_sBtnText := 'Start';

s_fbHmiBtnStateStop.p_eButtontype := E_HmiButtonType.PUSHBUTTON;
s_fbHmiBtnStateStop.p_bStaVisible := FALSE;
s_fbHmiBtnStateStop.p_bStaEnabled := FALSE;
s_fbHmiBtnStateStop.p_sBtnText := 'Stop';

s_fbHmiBtnStateReset.p_eButtontype := E_HmiButtonType.PUSHBUTTON;
s_fbHmiBtnStateReset.p_bStaVisible := FALSE;
s_fbHmiBtnStateReset.p_bStaEnabled := FALSE;
s_fbHmiBtnStateReset.p_sBtnText := 'Reset';

_m_Init := TRUE;
END_METHOD

METHOD PUBLIC m_Main : BOOL

IF NOT s_bInitDone THEN
	IF _m_Init() THEN 
		s_bInitDone := TRUE;
	END_IF
END_IF

_m_Devices();

m_Main := TRUE;
END_METHOD

PROPERTY PUBLIC p_eCtrlMode : E_CtrlMode
GET

p_eCtrlMode := s_eCtrlMode;
END_GET
END_PROPERTY

PROPERTY PUBLIC p_eCtrlState : E_CtrlState
GET

p_eCtrlState := s_eCtrlState;
END_GET
END_PROPERTY

END_FUNCTION_BLOCK

// ---- POUs/03 EM/FB_Interlock.TcPOU
FUNCTION_BLOCK FB_Interlock
VAR_INPUT
	i_bInterlocked : BOOL;
END_VAR
VAR
	s_bInterlocked : BOOL;
	s_sReason : STRING;
END_VAR


s_bInterlocked := i_bInterlocked;

PROPERTY PUBLIC p_bInterlocked : BOOL
GET

p_bInterlocked := s_bInterlocked;
END_GET
END_PROPERTY

PROPERTY PUBLIC p_sReason : STRING
GET

p_sReason := s_sReason;
END_GET
SET

s_sReason := p_sReason;
END_SET
END_PROPERTY

END_FUNCTION_BLOCK

// ---- POUs/03 EM/FB_InterlockHandler.TcPOU
FUNCTION_BLOCK FB_InterlockHandler
VAR_INPUT
	//--i_ref_stInterlockList : REFERENCE TO ST_InterlockList;
	i_stInterlockList : ST_InterlockList; 
END_VAR
VAR
	s_bInterlocked : BOOL;
	s_sReason : STRING(GVL.g_MAX_LEN_INTERLOCK_REASON);
	i : USINT;
	s_nInterlockCnt : USINT;
	
	s_ton : TON;
	s_nIndexShow : USINT := 0;
END_VAR


s_bInterlocked := FALSE;
s_sReason := '';
s_nInterlockCnt := 0;

//Old code showing only one (first found reson)
//--FOR i := 0 TO (GVL.g_LEN_INTERLOCK_LIST-1) DO
//--	IF i_stInterlockList.arr_Interlocks[i].bState THEN
//--		s_bInterlocked := i_stInterlockList.arr_Interlocks[i].bState;
//--		s_sReason := i_stInterlockList.arr_Interlocks[i].sReason;
//--		EXIT;
//--	END_IF
//--END_FOR

FOR i := 0 TO (GVL.g_LEN_INTERLOCK_LIST-1) DO
	IF i_stInterlockList.arr_Interlocks[i].bState THEN
		s_nInterlockCnt := s_nInterlockCnt + 1;
		s_bInterlocked := i_stInterlockList.arr_Interlocks[i].bState;
		//--s_sReason := i_stInterlockList.arr_Interlocks[i].sReason;
		IF s_nInterlockCnt > 1 THEN
			s_sReason := CONCAT(s_sReason, CONCAT('; ', i_stInterlockList.arr_Interlocks[i].sReason));
		ELSE
			s_sReason := i_stInterlockList.arr_Interlocks[i].sReason;
		END_IF	
	END_IF
END_FOR

//New code showing all active interlocks time based
(*
	s_ton(IN := NOT(s_ton.Q), PT := T#2S);

	IF s_ton.Q THEN
		IF i_stInterlockList.arr_Interlocks[s_nIndexShow].bState THEN
			s_bInterlocked := i_stInterlockList.arr_Interlocks[s_nIndexShow].bState;
			s_sReason := i_stInterlockList.arr_Interlocks[s_nIndexShow].sReason;
		END_IF
		
		IF s_nIndexShow < (GVL.g_LEN_INTERLOCK_LIST-1) THEN
			s_nIndexShow := s_nIndexShow + 1; 
		ELSE
			s_nIndexShow := 0;
		END_IF
		
	END_IF
*)

PROPERTY PUBLIC p_bInterlocked : BOOL
GET

p_bInterlocked := s_bInterlocked;
END_GET
END_PROPERTY

PROPERTY PUBLIC p_sReason : STRING
GET

p_sReason := s_sReason;
END_GET
END_PROPERTY

END_FUNCTION_BLOCK

// ---- POUs/FB_ModeStateControl_Base.TcPOU
FUNCTION_BLOCK FB_ModeStateControl_Base
VAR_INPUT
	i_bReqAutomatic : BOOL;
	i_bReqManual : BOOL;
	i_bReqMaintenance : BOOL;
	i_bReqIoTest : BOOL;
	i_bReqCleaning : BOOL;	

	i_bReqStart : BOOL;
	i_bReqStop : BOOL;
	i_bReqReset : BOOL;
	i_bStaStopped : BOOL;
END_VAR
VAR_OUTPUT
END_VAR
VAR
	s_bInitDone : BOOL := FALSE;	

	s_eCtrlMode : E_CtrlMode := E_CtrlMode.IDLE;
	s_eCtrlState : E_CtrlState := E_CtrlState.STOPPED;	
END_VAR

METHOD PRIVATE _m_Init : BOOL

//Mode buttons
s_fbHmiBtnModeAutomatic.p_eButtontype := E_HmiButtonType.PUSHBUTTON;
s_fbHmiBtnModeAutomatic.p_bStaVisible := FALSE;
s_fbHmiBtnModeAutomatic.p_bStaEnabled := FALSE;
s_fbHmiBtnModeAutomatic.p_sBtnText := 'Automatic';

s_fbHmiBtnModeManual.p_eButtontype := E_HmiButtonType.PUSHBUTTON;
s_fbHmiBtnModeManual.p_bStaVisible := FALSE;
s_fbHmiBtnModeManual.p_bStaEnabled := FALSE;
s_fbHmiBtnModeManual.p_sBtnText := 'Manual';

s_fbHmiBtnModeMaintenance.p_eButtontype := E_HmiButtonType.PUSHBUTTON;
s_fbHmiBtnModeMaintenance.p_bStaVisible := FALSE;
s_fbHmiBtnModeMaintenance.p_bStaEnabled := FALSE;
s_fbHmiBtnModeMaintenance.p_sBtnText := 'Maintenance';

s_fbHmiBtnModeIO.p_eButtontype := E_HmiButtonType.PUSHBUTTON;
s_fbHmiBtnModeIO.p_bStaVisible := FALSE;
s_fbHmiBtnModeIO.p_bStaEnabled := FALSE;
s_fbHmiBtnModeIO.p_sBtnText := 'IO';

s_fbHmiBtnModeCleaning.p_eButtontype := E_HmiButtonType.PUSHBUTTON;
s_fbHmiBtnModeCleaning.p_bStaVisible := FALSE;
s_fbHmiBtnModeCleaning.p_bStaEnabled := FALSE;
s_fbHmiBtnModeCleaning.p_sBtnText := 'Cleaning';

//State buttons
s_fbHmiBtnStateStart.p_eButtontype := E_HmiButtonType.PUSHBUTTON;
s_fbHmiBtnStateStart.p_bStaVisible := FALSE;
s_fbHmiBtnStateStart.p_bStaEnabled := FALSE;
s_fbHmiBtnStateStart.p_sBtnText := 'Start';

s_fbHmiBtnStateStop.p_eButtontype := E_HmiButtonType.PUSHBUTTON;
s_fbHmiBtnStateStop.p_bStaVisible := FALSE;
s_fbHmiBtnStateStop.p_bStaEnabled := FALSE;
s_fbHmiBtnStateStop.p_sBtnText := 'Stop';

s_fbHmiBtnStateReset.p_eButtontype := E_HmiButtonType.PUSHBUTTON;
s_fbHmiBtnStateReset.p_bStaVisible := FALSE;
s_fbHmiBtnStateReset.p_bStaEnabled := FALSE;
s_fbHmiBtnStateReset.p_sBtnText := 'Reset';

_m_Init := TRUE;
END_METHOD

METHOD PUBLIC m_Main : BOOL

IF (s_eCtrlState = E_CtrlState.IDLE) OR (s_eCtrlState = E_CtrlState.STOPPED) THEN
	IF i_bReqAutomatic THEN
		s_eCtrlMode := E_CtrlMode.AUTOMATIC;
	ELSIF i_bReqManual THEN
		s_eCtrlMode := E_CtrlMode.MANUAL;
	ELSIF i_bReqMaintenance THEN
		s_eCtrlMode := E_CtrlMode.MAINTENANCE;
	ELSIF i_bReqIoTest THEN
		s_eCtrlMode := E_CtrlMode.IO;
	ELSIF i_bReqCleaning THEN
		s_eCtrlMode := E_CtrlMode.CLEANING;
	END_IF
END_IF

CASE s_eCtrlMode OF
	E_CtrlMode.IDLE:
		;//Nothing
	
	E_CtrlMode.AUTOMATIC:
		m_ModeAutomatic();
	
	E_CtrlMode.MANUAL:
		m_ModeManual();
	
	E_CtrlMode.MAINTENANCE:
		m_ModeMaintenance();
	
	E_CtrlMode.IO:
		m_ModeIoTest();
		
	E_CtrlMode.CLEANING:
		m_ModeCleaning();
		
	ELSE
		s_eCtrlMode := E_CtrlMode.IDLE;
END_CASE

CASE s_eCtrlState OF
	E_CtrlState.STOPPED:
		m_StateStopped();
		
		IF i_bReqReset THEN
			s_eCtrlState := E_CtrlState.IDLE;
		END_IF	
		
	E_CtrlState.IDLE:
		m_StateIdle();
		
		IF i_bReqStop THEN
			s_eCtrlState := E_CtrlState.STOPPING;
		ELSIF i_bReqStart THEN
			s_eCtrlState := E_CtrlState.RUNNING;
		END_IF
	
	E_CtrlState.RUNNING:
		m_StateRunning();
		
		IF i_bReqStop THEN
			s_eCtrlState := E_CtrlState.STOPPING;
		END_IF
			
	E_CtrlState.STOPPING:
		m_StateStopping();
		
		IF i_bStaStopped THEN
			s_eCtrlState := E_CtrlState.STOPPED;
		END_IF
	
	ELSE
		s_eCtrlState := E_CtrlState.STOPPED;
END_CASE

m_Main := TRUE;
END_METHOD

METHOD PUBLIC m_ModeAutomatic : BOOL
END_METHOD

METHOD PUBLIC m_ModeCleaning : BOOL
END_METHOD

METHOD PUBLIC m_ModeIoTest : BOOL
END_METHOD

METHOD PUBLIC m_ModeMaintenance : BOOL
END_METHOD

METHOD PUBLIC m_ModeManual : BOOL
END_METHOD

METHOD PUBLIC m_StateIdle : BOOL
END_METHOD

METHOD PUBLIC m_StateRunning : BOOL
END_METHOD

METHOD PUBLIC m_StateStopped : BOOL
END_METHOD

METHOD PUBLIC m_StateStopping : BOOL
END_METHOD

END_FUNCTION_BLOCK

// ---- POUs/FB_InRange.TcPOU
FUNCTION_BLOCK FB_InRange
VAR_INPUT
	i_fValue : LREAL;
	i_fRange : LREAL;
END_VAR
VAR_OUTPUT
END_VAR
VAR
	nCntAuto : UINT;
	nCntManual : UINT;
	nCntMaintenance : UINT;
	
END_VAR


SUPER^.m_Main();

END_FUNCTION_BLOCK

// ---- GlobalTextList.TcGTLO
TEXTLIST GlobalTextList
  292 = '   Q      State     Error'
  1145 = '#s'
  593 = '%'
  744 = '%s'
  670 = 'Actual mode:'
  459 = 'Actual step Centering:'
  734 = 'Actual step Transport:'
  384 = 'Actual step:'
  659 = 'Actual step: %c'
  904 = 'Actual step: %s'
  858 = 'Air'
  1193 = 'Air pressure OK'
  961 = 'ALARM LIST'
  567 = 'Apply'
  838 = 'Automatic'
  503 = 'Backward'
  60 = 'Brake'
  947 = 'Brake Released'
  315 = 'Button 1'
  574 = 'Button 2'
  341 = 'BWD'
  784 = 'CCW'
  856 = 'Center'
  642 = 'Centering'
  857 = 'Centering position'
  67 = 'Centering TB'
  698 = 'Clamps lower closed'
  469 = 'Clamps lower opened'
  800 = 'Clamps upper closed'
  639 = 'Clamps upper opened'
  668 = 'Close'
  268 = 'Close Inner Door'
  269 = 'CM Docking Clamp Lower'
  647 = 'CM Docking Clamp Upper'
  14 = 'CM Door Opener'
  1012 = 'CM Door Shutter'
  117 = 'CM Pallet Centering'
  1154 = 'CM Pallet Conveyor'
  240 = 'CM Unlocking Pin Lower'
  71 = 'CM Unlocking Pin Upper'
  314 = 'Cmd     State     Error'
  271 = 'CW'
  736 = 'Dock TB'
  843 = 'Docking'
  379 = 'Docking Clamp Lower'
  767 = 'Docking Clamp Upper'
  316 = 'Docking Interface'
  621 = 'Docking position'
  866 = 'Docking Station'
  715 = 'Docking System'
  1135 = 'Door'
  638 = 'Door opened'
  281 = 'Door Opener'
  157 = 'Door Shutter'
  113 = 'Drive Error'
  342 = 'Drive Running'
  1278 = 'EM Docking Interface'
  299 = 'EM Pallet Centering'
  359 = 'EM Pallet Conveyor'
  364 = 'Err'
  979 = 'Erro'
  381 = 'Error'
  98 = 'Forward'
  324 = 'Front'
  782 = 'FWD'
  958 = 'High pressure'
  187 = 'Idle'
  439 = 'Infeed'
  114 = 'Infeed front'
  883 = 'Infeed front position'
  893 = 'Infeed rear'
  799 = 'Infeed rear position'
  376 = 'Left     Error'
  234 = 'Left     Right     Error'
  375 = 'Lock'
  192 = 'Main'
  848 = 'MainScreen'
  196 = 'Manual'
  445 = 'Motor'
  927 = 'Motor Stopped'
  675 = 'Motore'
  308 = 'Open'
  43 = 'Open Inner Door'
  104 = 'Opener almost closed'
  633 = 'Opener closed'
  769 = 'Opener opened'
  101 = 'Outer door opened'
  186 = 'Outer doorTB'
  674 = 'Outer TB'
  643 = 'Pallet Centering'
  933 = 'Pallet Conveyor'
  73 = 'Pallet Dectection'
  628 = 'Pallet Detection'
  254 = 'Pin lower locked'
  721 = 'Pin lower released'
  9 = 'Pin upper locked'
  677 = 'Pin upper released'
  693 = 'Power'
  115 = 'Power OK'
  276 = 'Q'
  387 = 'Q start/res'
  374 = 'Q start/reset'
  272 = 'qCCW'
  1022 = 'qCW'
  583 = 'qEnable'
  884 = 'Qrel'
  355 = 'Qrelay'
  172 = 'qRelay'
  49 = 'Qrelease'
  837 = 'Qreset'
  1180 = 'qReset'
  666 = 'Qrev'
  1008 = 'Qstart/reset'
  18 = 'Raw speed (Ai): %i'
  56 = 'Raw target speed (Ai): %i'
  796 = 'Raw target speed: %2.5f'
  812 = 'Raw target speed: %d4'
  270 = 'Raw target speed: %f1.1 mm/s'
  532 = 'Raw target speed: %f2 mm/s'
  112 = 'Raw target speed: %f3.1 mm/s'
  80 = 'Raw target speed: %i'
  623 = 'Raw target speed: %i mm/s'
  683 = 'Raw target speed: %i5'
  860 = 'Rear'
  952 = 'Release'
  783 = 'Released'
  258 = 'Reset'
  163 = 'Rest'
  888 = 'Reverse'
  813 = 'Run/Reset'
  1151 = 'Running'
  512 = 'Safety'
  697 = 'Safety OK'
  385 = 'sdf'
  703 = 'Shutter closed'
  510 = 'Shutter opened'
  944 = 'Speed'
  862 = 'Start / Reset'
  498 = 'State'
  322 = 'State     Error'
  616 = 'Stop'
  197 = 'Stopped'
  820 = 'Target speed: %i mm/s'
  393 = 'Target: %i mm/s'
  103 = 'TB to center'
  363 = 'TB to docking'
  537 = 'TB to Infeed'
  929 = 'Undock TB'
  1201 = 'Unlocking Pin Lower'
  474 = 'Unlocking Pin Upper'
  478 = 'Unlocking Pins Lower'
  255 = 'Unlocking Pins Upper'
  1088 = 'Utilities'
  896 = 'valve Error'
  1146 = 'Warning'
END_TEXTLIST
